{attribute 'qualified_only'}
{attribute 'strict'}
TYPE E_AlarmResponse :
(
	Abort_ImmediateError,
	Abort_Immediate,
	Stop_Immediate,
	Stop_Controlled,
	Hold_Immediate,
	Hold_Controlled,	
	Suspend_Immediate,
	Suspend_Controlled,
	NoResponse	
);
END_TYPE

(* stored: Version 1.1.0.1, ProductVersion 3.1.4024.9
   DUT E_AlarmResponse: Id {3cb16676-06c4-4bf3-9836-8856a06bd3ff} *)
